(* PLC project Unnamed, Unknown Unnamed 1 *)
(* stored: creationDateTime 2024-05-17T18:31:13, modificationDateTime 2024-05-17T18:44:05 *)

PROGRAM AND_NAND
  VAR
    INPUT_0 : BOOL;
    INPUT_1 : BOOL;
    INPUT_2 : BOOL;
    INPUT_3 : BOOL;
    OUTPUT_0 : BOOL;
    OUTPUT_1 : BOOL;
  END_VAR

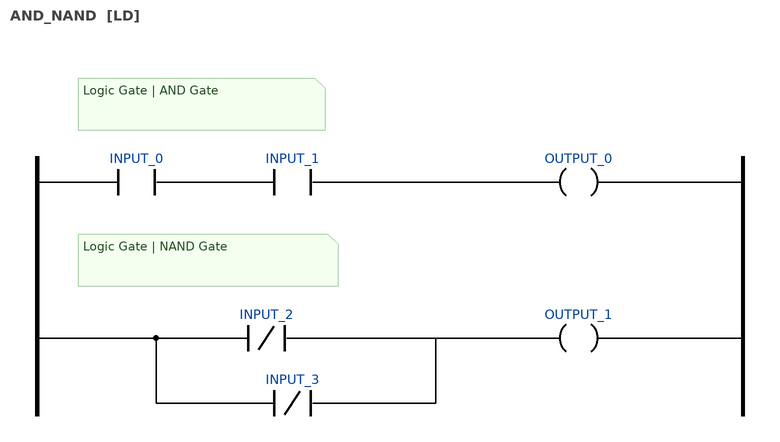
(* LD diagram, written out as Structured Text *)
(* Logic Gate | AND Gate *)
OUTPUT_0 := INPUT_0 AND INPUT_1;
(* Logic Gate | NAND Gate *)
OUTPUT_1 := NOT INPUT_2 OR NOT INPUT_3;
END_PROGRAM

CONFIGURATION Config0
  RESOURCE Res0 ON PLC
    TASK task0(INTERVAL := T#20ms, PRIORITY := 0);
    PROGRAM instance0 WITH task0 : AND_NAND;
  END_RESOURCE
END_CONFIGURATION
